// TIA Portal V17 export
// export: Created 2025-03-10T12:17:29.9811712Z, ExportSetting WithDefaults, DisplayName Totally Integrated Automation Portal, DisplayVersion V17 Update 8, DisplayName TIA Portal Openness, DisplayVersion V17 Update 8, DisplayName TIA Portal Version Control Interface, DisplayVersion V17, DisplayName SINAMICS Startdrive Advanced, DisplayVersion V17 SP2, DisplayName SINAMICS Startdrive G110M, G120, G120C, G120D, G120P, G115D, DisplayVersion V17 SP2, DisplayName SINAMICS Startdrive G130, G150, S120, S150, SINAMICS MV, S210, DisplayVersion V17 SP2, DisplayName STEP 7 Professional, DisplayVersion V17 Update 8, DisplayName SINUMERIK ONE STEP 7 Toolbox, DisplayVersion V17 Update 12, DisplayName SINUMERIK 840D sl STEP 7 Toolbox, DisplayVersion V17 Update 12, DisplayName STEP 7 Safety, DisplayVersion V17 Update 6, DisplayName WinCC Advanced, DisplayVersion V17 Update 8
VAR_GLOBAL   // PLC tag table "TEMPORAL_TAG_PANI"
   PART_PRESENT_SENSOR_UNIT_1 AT %MW5000 : Int;
   Delay_Z11_Start AT %T10 : Timer;
   Delay_Z21_Start AT %T20 : Timer;
   U01_STA4_BRUSH_WORN_ALARM AT %M100.0 : Bool;
   U01_STA4_BRUSH_WORN_INPUT AT %M100.1 : Bool;
   U01_STA4_BRUSH_CHANGE_ACK AT %M100.2 : Bool;
END_VAR
